// TwinCAT 3 PLC project L4_kolejiste
// ProgramVersion: 3.1.4026.21
// CompilerDefines: VISU_USEPROPERTYINFO
// libraries:
//   Tc2_Standard, * (Beckhoff Automation GmbH)
//   Tc2_System, * (Beckhoff Automation GmbH)
//   Tc3_Module, * (Beckhoff Automation GmbH)
//   VisuDialogs, * (System)
// project tree:
//   DUTs/ E_StateCmd.TcDUT (not stored), E_SystemState.TcDUT (not stored)
//   / GlobalTextList.TcGTLO, PlcTask.TcTTO
//   GVLs/ IO.TcGVL (not stored), TAGS.TcGVL (not stored), SCADA.TcGVL (not stored)
//   POUs/ FB_IO.TcPOU (not stored), FB_Barrier.TcPOU (not stored), FB_MachineControl.TcPOU (not stored), FB_State_Aborted.TcPOU, FB_State_Aborting.TcPOU, FB_State_Clearing.TcPOU (not stored), FB_State_Complete.TcPOU, FB_State_Completing.TcPOU (not stored), FB_State_Held.TcPOU, FB_State_Holding.TcPOU (not stored), FB_State_Manual.TcPOU (not stored), FB_State_Resuming.TcPOU, FB_State_Running.TcPOU, FB_State_Service.TcPOU (not stored), FB_State_Starting.TcPOU (not stored), FB_State_Stopped.TcPOU (not stored), FB_SwitchRouter.TcPOU (not stored), FB_DriveCtrl.TcPOU (not stored), MAIN.TcPOU (not stored)
//   VISUs/ Visualization.TcVIS
// real-time tasks:
//   TASK PlcTask: cycle T#10ms, priority 20, ADS port 350
//   TASK PlcTask1: cycle T#10ms, priority 21, ADS port 351
//   TASK PlcTask2: cycle T#10ms, priority 22, ADS port 352
//   TASK PlcTask3: cycle T#10ms, priority 23, ADS port 353
// I/O:
//   DEVICE Device 2 (EtherCAT), AmsNetId 169.254.109.136.3.1
//     Term 23 (EK1100) [EK1100 EtherCAT Coupler (2A E-Bus)]
//       Term 24 (EL1008) [EL1008 8Ch. Dig. Input 24V, 3ms]
//       Term 25 (EL1008) [EL1008 8Ch. Dig. Input 24V, 3ms]
//       Term 26 (EL2008) [EL2008 8Ch. Dig. Output 24V, 0.5A]
//       Term 29 (EL9011) [EL9011 End Terminal]
// variable links:
//   (this object) <-> Device 2 (EtherCAT)/Term 23 (EK1100)/Term 24 (EL1008)
//     PlcTask Inputs/IO.DI{0..7} <-> Channel {1..8}/Input  (8 links)
//     PlcTask Inputs/TAGS.PRE_I <-> Channel 4/Input
//     PlcTask Inputs/TAGS.PRE_II <-> Channel 5/Input
//     PlcTask Inputs/TAGS.PRE_KLA <-> Channel 4/Input
//     PlcTask Inputs/TAGS.PRE_OPA <-> Channel 5/Input
//     PlcTask Inputs/TAGS.TLA_LEV <-> Channel 6/Input
//     PlcTask Inputs/TAGS.TLA_PRA <-> Channel 7/Input
//     PlcTask Inputs/TAGS.TLA_ZAD <-> Channel 8/Input
//     PlcTask Inputs/TAGS.VYH_LEV <-> Channel 1/Input
//     PlcTask Inputs/TAGS.VYH_PRA <-> Channel 2/Input
//     PlcTask Inputs/TAGS.VYH_ZAD <-> Channel 3/Input
//   (this object) <-> Device 2 (EtherCAT)/Term 23 (EK1100)/Term 25 (EL1008)
//     PlcTask Inputs/IO.DI{8..11} <-> Channel {1..4}/Input  (4 links)
//     PlcTask Inputs/TAGS.HRA_LEV <-> Channel 2/Input
//     PlcTask Inputs/TAGS.HRA_PRA <-> Channel 1/Input
//     PlcTask Inputs/TAGS.HRA_ZAD <-> Channel 3/Input
//     PlcTask Inputs/TAGS.HRA_ZAV <-> Channel 4/Input
//     PlcTask Inputs/TAGS.SP1 <-> Channel 2/Input
//     PlcTask Inputs/TAGS.SP2 <-> Channel 4/Input
//   (this object) <-> Device 2 (EtherCAT)/Term 23 (EK1100)/Term 26 (EL2008)
//     PlcTask Outputs/TAGS.IMP_LEV <-> Channel 4/Output
//     PlcTask Outputs/TAGS.IMP_PRA <-> Channel 5/Output
//     PlcTask Outputs/TAGS.IMP_ZAD <-> Channel 6/Output
//     PlcTask Outputs/TAGS.JIZDA <-> Channel 8/Output
//     PlcTask Outputs/TAGS.KLADNY <-> Channel 2/Output
//     PlcTask Outputs/TAGS.OPACNY <-> Channel 3/Output
//     PlcTask Outputs/TAGS.VYHYBKY <-> Channel 7/Output
//     PlcTask Outputs/TAGS.ZAVORY <-> Channel 1/Output

CONFIGURATION L4_kolejiste
    RESOURCE PLC ON TwinCAT3
        TASK PlcTask(INTERVAL := T#10ms, PRIORITY := 23);
        PROGRAM MAIN WITH PlcTask : MAIN;
    END_RESOURCE
END_CONFIGURATION

// ---- POUs/FB_State_Aborted.TcPOU
// State handler: ABORTED
// Holds fault flag. Waits for RESET edge AND E-STOP safe → CLEARING.
FUNCTION_BLOCK FB_State_Aborted
VAR_INPUT
    bExecute        : BOOL;
    bReset          : BOOL;   // Edge from MachineControl
    bEStop_Safe     : BOOL;   // TRUE = no E-STOP active
END_VAR
VAR_OUTPUT
    outCmd          : E_StateCmd := E_StateCmd.NONE;
    outEnable_Auto  : BOOL;
    outEnable_Man   : BOOL;
    outgvFault      : BOOL;
    outInit_VYHYBKY : BOOL;
    outInit_IMP_LEV : BOOL;
    outInit_IMP_PRA : BOOL;
END_VAR

IF NOT bExecute THEN
    outCmd          := E_StateCmd.NONE;
    outEnable_Auto  := FALSE;
    outEnable_Man   := FALSE;
    outgvFault      := FALSE;
    outInit_VYHYBKY := FALSE;
    outInit_IMP_LEV := FALSE;
    outInit_IMP_PRA := FALSE;
    RETURN;
END_IF

outEnable_Auto  := FALSE;
outEnable_Man   := FALSE;
outgvFault      := TRUE;   // Keep fault flag active while aborted
outInit_VYHYBKY := FALSE;
outInit_IMP_LEV := FALSE;
outInit_IMP_PRA := FALSE;

IF bReset AND bEStop_Safe THEN
    outCmd := E_StateCmd.TO_CLEARING;
ELSE
    outCmd := E_StateCmd.NONE;
END_IF

END_FUNCTION_BLOCK

// ---- POUs/FB_State_Aborting.TcPOU
// State handler: ABORTING
// Transient state — raises fault flag and immediately signals → ABORTED.
// Add safe-stop sequencing here if needed.
FUNCTION_BLOCK FB_State_Aborting
VAR_INPUT
    bExecute    : BOOL;
END_VAR
VAR_OUTPUT
    outCmd          : E_StateCmd := E_StateCmd.NONE;
    outEnable_Auto  : BOOL;
    outEnable_Man   : BOOL;
    outgvFault      : BOOL;
    outInit_VYHYBKY : BOOL;
    outInit_IMP_LEV : BOOL;
    outInit_IMP_PRA : BOOL;
END_VAR

IF NOT bExecute THEN
    outCmd          := E_StateCmd.NONE;
    outEnable_Auto  := FALSE;
    outEnable_Man   := FALSE;
    outgvFault      := FALSE;
    outInit_VYHYBKY := FALSE;
    outInit_IMP_LEV := FALSE;
    outInit_IMP_PRA := FALSE;
    RETURN;
END_IF

outEnable_Auto  := FALSE;
outEnable_Man   := FALSE;
outgvFault      := TRUE;   // Fault active during abort
outInit_VYHYBKY := FALSE;
outInit_IMP_LEV := FALSE;
outInit_IMP_PRA := FALSE;

// Immediate transition
outCmd := E_StateCmd.TO_ABORTED;

END_FUNCTION_BLOCK

// ---- POUs/FB_State_Complete.TcPOU
// State handler: COMPLETE
// Waits for RESET edge → STOPPED.
FUNCTION_BLOCK FB_State_Complete
VAR_INPUT
    bExecute    : BOOL;
    bReset      : BOOL;   // Edge from MachineControl
END_VAR
VAR_OUTPUT
    outCmd          : E_StateCmd := E_StateCmd.NONE;
    outEnable_Auto  : BOOL;
    outEnable_Man   : BOOL;
    outgvFault      : BOOL;
    outInit_VYHYBKY : BOOL;
    outInit_IMP_LEV : BOOL;
    outInit_IMP_PRA : BOOL;
END_VAR

IF NOT bExecute THEN
    outCmd          := E_StateCmd.NONE;
    outEnable_Auto  := FALSE;
    outEnable_Man   := FALSE;
    outgvFault      := FALSE;
    outInit_VYHYBKY := FALSE;
    outInit_IMP_LEV := FALSE;
    outInit_IMP_PRA := FALSE;
    RETURN;
END_IF

outEnable_Auto  := FALSE;
outEnable_Man   := FALSE;
outgvFault      := FALSE;
outInit_VYHYBKY := FALSE;
outInit_IMP_LEV := FALSE;
outInit_IMP_PRA := FALSE;

IF bReset THEN
    outCmd := E_StateCmd.TO_STOPPED;
ELSE
    outCmd := E_StateCmd.NONE;
END_IF

END_FUNCTION_BLOCK

// ---- POUs/FB_State_Held.TcPOU
// State handler: HELD
// Waits for START edge → RESUMING, or MAN edge → MANUAL.
FUNCTION_BLOCK FB_State_Held
VAR_INPUT
    bExecute    : BOOL;
    bStart      : BOOL;   // Edge from MachineControl
    bMan        : BOOL;   // Edge from MachineControl
END_VAR
VAR_OUTPUT
    outCmd          : E_StateCmd := E_StateCmd.NONE;
    outEnable_Auto  : BOOL;
    outEnable_Man   : BOOL;
    outgvFault      : BOOL;
    outInit_VYHYBKY : BOOL;
    outInit_IMP_LEV : BOOL;
    outInit_IMP_PRA : BOOL;
END_VAR

IF NOT bExecute THEN
    outCmd          := E_StateCmd.NONE;
    outEnable_Auto  := FALSE;
    outEnable_Man   := FALSE;
    outgvFault      := FALSE;
    outInit_VYHYBKY := FALSE;
    outInit_IMP_LEV := FALSE;
    outInit_IMP_PRA := FALSE;
    RETURN;
END_IF

outEnable_Auto  := FALSE;
outEnable_Man   := FALSE;
outgvFault      := FALSE;
outInit_VYHYBKY := FALSE;
outInit_IMP_LEV := FALSE;
outInit_IMP_PRA := FALSE;

IF bStart THEN
    outCmd := E_StateCmd.TO_RESUMING;
ELSIF bMan THEN
    outCmd := E_StateCmd.TO_MANUAL;
ELSE
    outCmd := E_StateCmd.NONE;
END_IF

END_FUNCTION_BLOCK

// ---- POUs/FB_State_Resuming.TcPOU
// State handler: RESUMING
// Transient state — immediately signals → RUNNING.
// Add ramp-up logic here if needed in the future.
FUNCTION_BLOCK FB_State_Resuming
VAR_INPUT
    bExecute    : BOOL;
END_VAR
VAR_OUTPUT
    outCmd          : E_StateCmd := E_StateCmd.NONE;
    outEnable_Auto  : BOOL;
    outEnable_Man   : BOOL;
    outgvFault      : BOOL;
    outInit_VYHYBKY : BOOL;
    outInit_IMP_LEV : BOOL;
    outInit_IMP_PRA : BOOL;
END_VAR

IF NOT bExecute THEN
    outCmd          := E_StateCmd.NONE;
    outEnable_Auto  := FALSE;
    outEnable_Man   := FALSE;
    outgvFault      := FALSE;
    outInit_VYHYBKY := FALSE;
    outInit_IMP_LEV := FALSE;
    outInit_IMP_PRA := FALSE;
    RETURN;
END_IF

outEnable_Auto  := FALSE;
outEnable_Man   := FALSE;
outgvFault      := FALSE;
outInit_VYHYBKY := FALSE;
outInit_IMP_LEV := FALSE;
outInit_IMP_PRA := FALSE;

// Immediate transition
outCmd := E_StateCmd.TO_RUNNING;

END_FUNCTION_BLOCK

// ---- POUs/FB_State_Running.TcPOU
// State handler: RUNNING
// Auto sequence enabled. STOP edge → COMPLETING. MAN edge → HOLDING.
FUNCTION_BLOCK FB_State_Running
VAR_INPUT
    bExecute    : BOOL;
    bStop       : BOOL;   // Edge from MachineControl
    bMan        : BOOL;   // Edge from MachineControl
END_VAR
VAR_OUTPUT
    outCmd          : E_StateCmd := E_StateCmd.NONE;
    outEnable_Auto  : BOOL;
    outEnable_Man   : BOOL;
    outgvFault      : BOOL;
    outInit_VYHYBKY : BOOL;
    outInit_IMP_LEV : BOOL;
    outInit_IMP_PRA : BOOL;
END_VAR

IF NOT bExecute THEN
    outCmd          := E_StateCmd.NONE;
    outEnable_Auto  := FALSE;
    outEnable_Man   := FALSE;
    outgvFault      := FALSE;
    outInit_VYHYBKY := FALSE;
    outInit_IMP_LEV := FALSE;
    outInit_IMP_PRA := FALSE;
    RETURN;
END_IF

outEnable_Auto  := TRUE;
outEnable_Man   := FALSE;
outgvFault      := FALSE;
outInit_VYHYBKY := FALSE;
outInit_IMP_LEV := FALSE;
outInit_IMP_PRA := FALSE;

IF bStop THEN
    outCmd := E_StateCmd.TO_COMPLETING;
ELSIF bMan THEN
    outCmd := E_StateCmd.TO_HOLDING;
ELSE
    outCmd := E_StateCmd.NONE;
END_IF

END_FUNCTION_BLOCK

// ---- GlobalTextList.TcGTLO
TEXTLIST GlobalTextList
  851 = 'ABORTED'
  620 = 'CLEARING'
  335 = 'COMPLETE'
  790 = 'COMPLETE. Press Reset'
  183 = 'Estop'
  598 = 'HELD'
  997 = 'Jizda klad'
  36 = 'Jizda opa'
  670 = 'Man'
  125 = 'MANUAL'
  597 = 'Reset'
  374 = 'Running'
  463 = 'Start'
  414 = 'STARTING'
  748 = 'Stop'
  920 = 'STOPPED'
  977 = 'vyh leva'
  696 = 'vyh prava'
  277 = 'vyh zadni'
  373 = 'zavora'
END_TEXTLIST

// ---- VISUs/Visualization.TcVIS
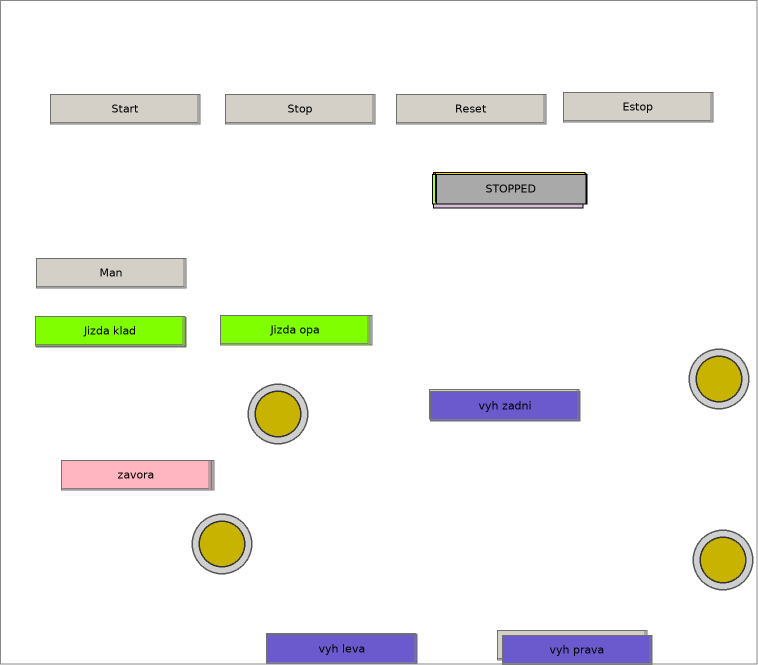
VISUALIZATION Visualization  // 758x665
    Button (50,94 150x30), "Start"
        tap SCADA.SCADA_START
    Button (225,94 150x30), "Stop"
        tap SCADA.SCADA_STOP
    Button (36,258 150x30), "Man", input disabled if: SCADA.systemstav=11
        tap SCADA.SCADA_MAN
    Button (396,94 150x30), "Reset"
        tap SCADA.SCADA_RESET
    Button (36,317 150x30), "Jizda klad", input disabled if: SCADA.systemstav<>11
        toggle SCADA.SCADA_MAN_OPACNY
    Button (64,460 150x30), "zavora", input disabled if: SCADA.systemstav<>11
        OnMouseClick: toggle SCADA.SCADA_MAN_ZAVORY
    Button (497,630 150x30), "vyh prava", input disabled if: SCADA.systemstav<>11
        tap SCADA.SCADA_MAN_IMP_PRA
    Button (429,389 150x30), "vyh zadni", input disabled if: SCADA.systemstav<>11
        tap SCADA.SCADA_MAN_IMP_ZAD
    Button (266,633 150x30), "vyh leva", input disabled if: SCADA.systemstav<>11
        tap SCADA.SCADA_MAN_IMP_LEV
    Button (222,315 150x30), "Jizda opa", input disabled if: SCADA.systemstav<>11
        toggle SCADA.SCADA_MAN_KLADNY
    Button (563,92 150x30), "Estop"
        toggle SCADA.SCADA_ESTOP
    Lamp1 (243,379 70x70), variable: TAGS.HRA_ZAV, style: Lamp-Lamp1-Yellow
    Lamp1 (187,509 70x70), variable: TAGS.HRA_LEV, style: Lamp-Lamp1-Yellow
    Lamp1 (688,525 70x70), variable: TAGS.HRA_PRA, style: Lamp-Lamp1-Yellow
    Lamp1 (684,344 70x70), variable: TAGS.HRA_ZAD, style: Lamp-Lamp1-Yellow
    Rectangle (436,173 150x30), "MANUAL", text variable: SCADA.systemstav, invisible if: SCADA.systemstav<>11
    Rectangle (433,178 150x30), "CLEARING", text variable: SCADA.systemstav, invisible if: SCADA.systemstav<>10
    Rectangle (433,172 150x30), "ABORTED", text variable: SCADA.systemstav, invisible if: SCADA.systemstav<>9
    Rectangle (435,173 150x30), "COMPLETE. Press Reset", text variable: SCADA.systemstav, invisible if: SCADA.systemstav<>7
    Rectangle (437,174 150x30), "HELD", text variable: SCADA.systemstav, invisible if: SCADA.systemstav<>4
    Rectangle (432,174 150x30), "Running", text variable: SCADA.systemstav, invisible if: SCADA.systemstav<>2
    Rectangle (435,172 150x30), "STARTING", text variable: SCADA.systemstav, invisible if: SCADA.systemstav<>1
    Rectangle (436,174 150x30), "STOPPED", text variable: SCADA.systemstav, invisible if: SCADA.systemstav<>0
    Button (35,316 150x30), "Jizda klad", invisible if: NOT MAIN.fbDrive.outKLADNY
        toggle SCADA.SCADA_MAN_OPACNY
    Button (220,315 150x30), "Jizda opa", invisible if: NOT MAIN.fbDrive.outOPACNY
        toggle SCADA.SCADA_MAN_KLADNY
    Button (61,460 150x30), "zavora", invisible if: NOT TAGS.ZAVORY, input disabled if: SCADA.systemstav<>11
        OnMouseClick: toggle SCADA.SCADA_MAN_ZAVORY
    Button (267,634 150x30), "vyh leva", invisible if: NOT TAGS.VYH_LEV, input disabled if: SCADA.systemstav<>11
        tap SCADA.SCADA_MAN_IMP_LEV
    Button (502,635 150x30), "vyh prava", invisible if: NOT TAGS.VYH_PRA, input disabled if: SCADA.systemstav<>11
        tap SCADA.SCADA_MAN_IMP_PRA
    Button (430,391 150x30), "vyh zadni", invisible if: NOT TAGS.VYH_ZAD, input disabled if: SCADA.systemstav<>11
        tap SCADA.SCADA_MAN_IMP_ZAD
END_VISUALIZATION
